// SIMATIC STEP 7 (V5.x) project hello_world
// CPU: CPU 313C
// CPU: CPU 313C
// station: Hardware
// station: SIMATIC 300(2)
// station: P_ADR_BUS
// station: Hardware
// station: SIMATIC 300(1)
// station: P_ADR_BUS
// program: S7 Program(1)
// program: S7 Program(2)

ORGANIZATION_BLOCK OB 1
TITLE = "Main Program Sweep (Cycle)"
VERSION : 0.1
VAR_TEMP
  OB1_EV_CLASS : BYTE ;	//Bits 0-3 = 1 (Coming event), Bits 4-7 = 1 (Event class 1)
  OB1_SCAN_1 : BYTE ;	//1 (Cold restart scan 1 of OB 1), 3 (Scan 2-n of OB 1)
  OB1_PRIORITY : BYTE ;	//Priority of OB Execution
  OB1_OB_NUMBR : BYTE ;	//1 (Organization block 1, OB1)
  OB1_RESERVED_1 : BYTE ;	//Reserved for system
  OB1_RESERVED_2 : BYTE ;	//Reserved for system
  OB1_PREV_CYCLE : INT ;	//Cycle time of previous OB1 scan (milliseconds)
  OB1_MIN_CYCLE : INT ;	//Minimum cycle time of OB1 (milliseconds)
  OB1_MAX_CYCLE : INT ;	//Maximum cycle time of OB1 (milliseconds)
  OB1_DATE_TIME : DATE_AND_TIME ;	//Date and time OB1 started
END_VAR
BEGIN
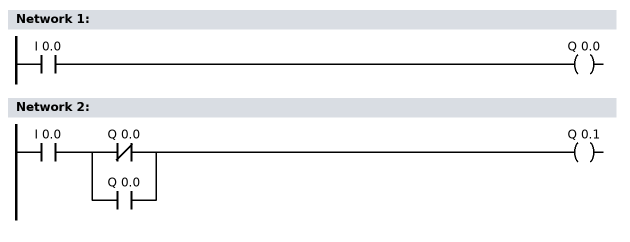
NETWORK
TITLE =
      A     I 0.0;
      =     Q 0.0;
NETWORK
TITLE =
      A     I 0.0;
      A(;
      ON    Q 0.0;
      O     Q 0.0;
      );
      =     Q 0.1;
END_ORGANIZATION_BLOCK

ORGANIZATION_BLOCK OB 1
TITLE = "Main Program Sweep (Cycle)"
VERSION : 0.1
VAR_TEMP
  OB1_EV_CLASS : BYTE ;	//Bits 0-3 = 1 (Coming event), Bits 4-7 = 1 (Event class 1)
  OB1_SCAN_1 : BYTE ;	//1 (Cold restart scan 1 of OB 1), 3 (Scan 2-n of OB 1)
  OB1_PRIORITY : BYTE ;	//Priority of OB Execution
  OB1_OB_NUMBR : BYTE ;	//1 (Organization block 1, OB1)
  OB1_RESERVED_1 : BYTE ;	//Reserved for system
  OB1_RESERVED_2 : BYTE ;	//Reserved for system
  OB1_PREV_CYCLE : INT ;	//Cycle time of previous OB1 scan (milliseconds)
  OB1_MIN_CYCLE : INT ;	//Minimum cycle time of OB1 (milliseconds)
  OB1_MAX_CYCLE : INT ;	//Maximum cycle time of OB1 (milliseconds)
  OB1_DATE_TIME : DATE_AND_TIME ;	//Date and time OB1 started
END_VAR
BEGIN
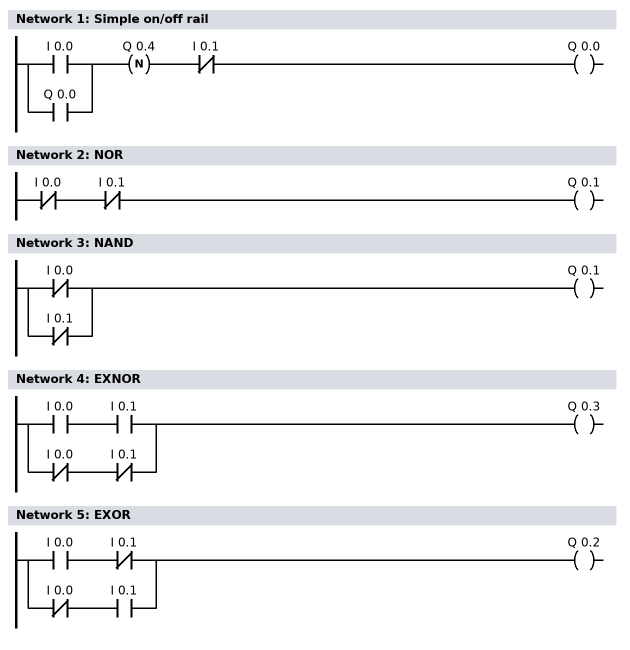
NETWORK
TITLE = Simple on/off rail
      A(;
      O     I 0.0;
      O     Q 0.0;
      );
      FN    Q 0.4;
      AN    I 0.1;
      =     Q 0.0;
NETWORK
TITLE = NOR
      AN    I 0.0;
      AN    I 0.1;
      =     Q 0.1;
NETWORK
TITLE = NAND
      ON    I 0.0;
      ON    I 0.1;
      =     Q 0.1;
NETWORK
TITLE = EXNOR
      A     I 0.0;
      A     I 0.1;
      O;
      AN    I 0.0;
      AN    I 0.1;
      =     Q 0.3;
NETWORK
TITLE = EXOR
      A     I 0.0;
      AN    I 0.1;
      O;
      AN    I 0.0;
      A     I 0.1;
      =     Q 0.2;
END_ORGANIZATION_BLOCK
